% RSLogix 500 project PROJECT2.RSS, saved by version 8.30.00.16 %
PROJECT "PROJECT2"    % processor: Bul.1763 MicroLogix 1100 Series B %

PROGRAM FILES
  LAD 2 "MAIN"  4 rungs
  LAD 3 "DIGITAL IO"  8 rungs
  LAD 4 "CONTROLS"  5 rungs

DATA FILES
  O0 OUTPUT  4 elements
  I1 INPUT  6 elements
  S2 STATUS  66 elements
  B3 BINARY  1 elements
  T4 TIMER  1 elements
  C5 COUNTER  1 elements
  R6 CONTROL  1 elements
  N7 INTEGER  1 elements
  F8 FLOAT  1 elements

LADDER 2 "MAIN"
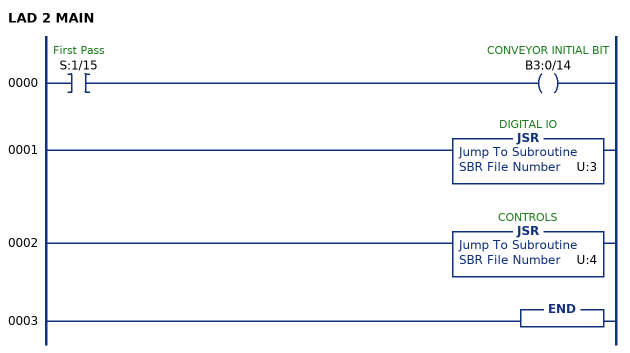
% Rung: 0 %
SOR XIC S:1/15 OTE B3:0/14 EOR
%   S:1/15  "First Pass" %
%   B3:0/14  "CONVEYOR INITIAL BIT" %
% Rung: 1 %
SOR JSR U:3 EOR
%   U:3  "DIGITAL IO" %
% Rung: 2 %
SOR JSR U:4 EOR
%   U:4  "CONTROLS" %
% Rung: 3 %
SOR END EOR

LADDER 3 "DIGITAL IO"
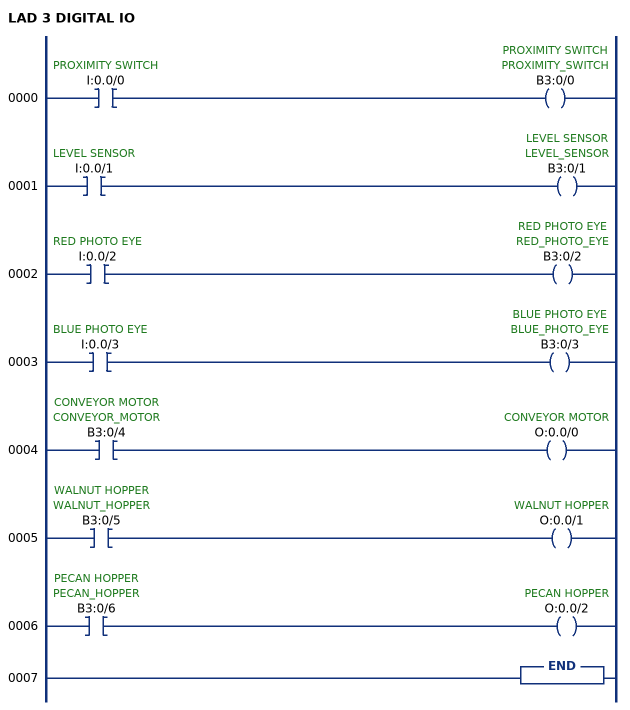
% Rung: 0 %
SOR XIC I:0.0/0 OTE B3:0/0 EOR
%   I:0.0/0  "PROXIMITY SWITCH" %
%   B3:0/0  PROXIMITY_SWITCH  "PROXIMITY SWITCH" %
% Rung: 1 %
SOR XIC I:0.0/1 OTE B3:0/1 EOR
%   I:0.0/1  "LEVEL SENSOR" %
%   B3:0/1  LEVEL_SENSOR  "LEVEL SENSOR" %
% Rung: 2 %
SOR XIC I:0.0/2 OTE B3:0/2 EOR
%   I:0.0/2  "RED PHOTO EYE" %
%   B3:0/2  RED_PHOTO_EYE  "RED PHOTO EYE" %
% Rung: 3 %
SOR XIC I:0.0/3 OTE B3:0/3 EOR
%   I:0.0/3  "BLUE PHOTO EYE" %
%   B3:0/3  BLUE_PHOTO_EYE  "BLUE PHOTO EYE" %
% Rung: 4 %
SOR XIC B3:0/4 OTE O:0.0/0 EOR
%   B3:0/4  CONVEYOR_MOTOR  "CONVEYOR MOTOR" %
%   O:0.0/0  "CONVEYOR MOTOR" %
% Rung: 5 %
SOR XIC B3:0/5 OTE O:0.0/1 EOR
%   B3:0/5  WALNUT_HOPPER  "WALNUT HOPPER" %
%   O:0.0/1  "WALNUT HOPPER" %
% Rung: 6 %
SOR XIC B3:0/6 OTE O:0.0/2 EOR
%   B3:0/6  PECAN_HOPPER  "PECAN HOPPER" %
%   O:0.0/2  "PECAN HOPPER" %
% Rung: 7 %
SOR END EOR

LADDER 4 "CONTROLS"
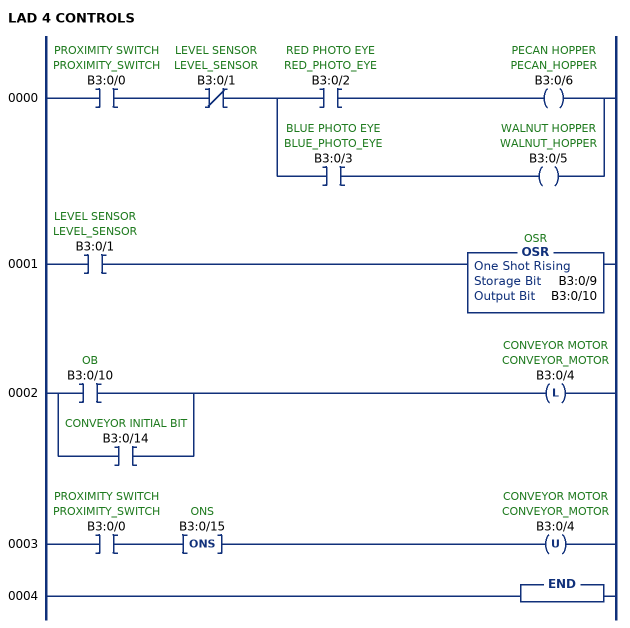
% Rung: 0 %
SOR XIC B3:0/0 XIO B3:0/1 BST XIC B3:0/2 OTE B3:0/6 NXB XIC B3:0/3 OTE B3:0/5 BND EOR
%   B3:0/0  PROXIMITY_SWITCH  "PROXIMITY SWITCH" %
%   B3:0/1  LEVEL_SENSOR  "LEVEL SENSOR" %
%   B3:0/2  RED_PHOTO_EYE  "RED PHOTO EYE" %
%   B3:0/6  PECAN_HOPPER  "PECAN HOPPER" %
%   B3:0/3  BLUE_PHOTO_EYE  "BLUE PHOTO EYE" %
%   B3:0/5  WALNUT_HOPPER  "WALNUT HOPPER" %
% Rung: 1 %
SOR XIC B3:0/1 OSR B3:0/9 B3:0/10 EOR
%   B3:0/1  LEVEL_SENSOR  "LEVEL SENSOR" %
%   B3:0/9  "OSR" %
%   B3:0/10  "OB" %
% Rung: 2 %
SOR BST XIC B3:0/10 NXB XIC B3:0/14 BND OTL B3:0/4 EOR
%   B3:0/10  "OB" %
%   B3:0/14  "CONVEYOR INITIAL BIT" %
%   B3:0/4  CONVEYOR_MOTOR  "CONVEYOR MOTOR" %
% Rung: 3 %
SOR XIC B3:0/0 ONS B3:0/15 OTU B3:0/4 EOR
%   B3:0/0  PROXIMITY_SWITCH  "PROXIMITY SWITCH" %
%   B3:0/15  "ONS" %
%   B3:0/4  CONVEYOR_MOTOR  "CONVEYOR MOTOR" %
% Rung: 4 %
SOR END EOR

OTHER DOCUMENTED ADDRESSES
  B3:0/7  "PROXIMITY SWITCH ENERGIZE BIT"
  B3:0/8  "ONS"
  B3:0/11  "WALNUT SB"
  B3:0/12  "WALNUT OB"
  B3:0/13  "CONVEYOR CONTROL BIT"
